// TwinCAT 3 PLC project CX5240
// ProgramVersion: 3.1.4026.13
// libraries:
//   CmpBitmapPool, * (System)
//   Tc2_Standard, * (Beckhoff Automation GmbH)
//   Tc2_System, * (Beckhoff Automation GmbH)
//   Tc3_Module, * (Beckhoff Automation GmbH)
//   VisuDialogs, * (System)
//   VisuSymbols,3.5.10.0,System
// project tree:
//   Enums/ E_Status.TcDUT (not stored)
//   Function Blocks/ FB_AnalogInputScaling.TcPOU (not stored), FB_DisplacementControl.TcPOU (not stored), FB_Encoder.TcPOU (not stored), FB_Integrator.TcPOU, FB_Joystick.TcPOU (not stored), FB_JoystickInputScaling.TcPOU (not stored), FB_DisplacementValveOutput.TcPOU (not stored), FB_StartPos.TcPOU, FB_YokeInputScaling.TcPOU (not stored), FB_ValveOutput.TcPOU
//   / GlobalTextList.TcGTLO (not stored), PlcTask.TcTTO (not stored)
//   GVLs/ G_IO.TcGVL (not stored), G_Parameters.TcGVL (not stored), G_Sensors.TcGVL (not stored), HMI.TcGVL
//   POUs/ MAIN.TcPOU, P_Inputs.TcPOU (not stored), P_MotionControl.TcPOU (not stored), P_Outputs.TcPOU
//   Struct/ ST_AnalogInputScaling.TcDUT (not stored), ST_JoystickInputScaling.TcDUT, ST_YokeInputScaling.TcDUT (not stored), ST_Parameters.TcDUT, ST_ValveDeadBand.TcDUT (not stored), ST_ValveOutput.TcDUT (not stored)
// real-time tasks:
//   TASK PlcTask: cycle T#1ms, priority 20, ADS port 350
//   TASK VISU_TASK: cycle T#200000us, priority 30, ADS port 351
// I/O:
//   DEVICE Device 1 (EtherCAT), AmsNetId 128.39.200.126.2.1
//     Term 1 (EK1200) [EK1200-5000 EtherCAT Power supply (2A E-Bus)]
//       Term 2 (EL1859) [EL1859 8Ch. Dig. Input 24V, 3ms, 8Ch. Dig. Output 24V, 0.5A]
//       Term 3 (EL3174) [EL3174 4Ch. Ana. Input +/-10V Diff., +/-20mA SingleEnded, 16 Bit]
//       Term 4 (EL4032) [EL4032 2Ch. Ana. Output +/-10V, 12bit]
//       Term 7 (EL3204) [EL3204 4Ch. Ana. Input PT100 (RTD)]
//       Term 8 (EK1110) [EK1110 EtherCAT extension]
//     Term 14 (EK1818) [EK1818 EtherCAT IO-Coupler  (1A E-Bus, 8 Ch. Dig. In, 3ms, 4 Ch. Dig. Out 24V, 0,5A)] (disabled)
//       Term 10 (EL1008) [EL1008 8Ch. Dig. Input 24V, 3ms]
//       Term 11 (EL3174) [EL3174 4Ch. Ana. Input +/-10V Diff., +/-20mA SingleEnded, 16 Bit]
//       Term 12 (EL3068) [EL3068 8Ch. Ana. Input 0-10V]
//       Term 5 (EL4032) [EL4032 2Ch. Ana. Output +/-10V, 12bit]
//       Term 6 (EL4122) [EL4122 2Ch. Ana. Output  4-20mA, 16bit]
//       Term 17 (EL9011) [EL9011 End Terminal]
//     Box 13 (Fraba EtherCAT) [Absolute Rotary Encoder IXARC V01.05] (disabled)
// variable links:
//   CX5240/CX5240 Instance <-> Device 1 (EtherCAT)/Term 1 (EK1200)/Term 2 (EL1859)
//     PlcTask Inputs/G_IO.bTestNew <-> Channel 1/Input
//   CX5240/CX5240 Instance <-> Device 1 (EtherCAT)/Term 14 (EK1818)
//     PlcTask Inputs/G_IO.bEmgOk <-> Channel 1/Input
//     PlcTask Outputs/G_IO.bEnablePCDV <-> Channel 10/Output
//     PlcTask Outputs/G_IO.bOpenBrakes <-> Channel 9/Output
//     PlcTask Outputs/G_IO.bWinchValveEnable <-> Channel 11/Output
//   CX5240/CX5240 Instance <-> Device 1 (EtherCAT)/Term 14 (EK1818)/Term 10 (EL1008)
//     PlcTask Inputs/G_IO.bAutoSwtich <-> Channel 3/Input
//     PlcTask Inputs/G_IO.bDisplacementEnable <-> Channel 7/Input
//     PlcTask Inputs/G_IO.bManualSwtich <-> Channel 1/Input
//     PlcTask Inputs/G_IO.bOffSwtich <-> Channel 2/Input
//     PlcTask Inputs/G_IO.bStartButton <-> Channel 4/Input
//     PlcTask Inputs/G_IO.bStopButton <-> Channel 5/Input
//     PlcTask Inputs/G_IO.bWinchEnable <-> Channel 6/Input
//   CX5240/CX5240 Instance <-> Device 1 (EtherCAT)/Term 14 (EK1818)/Term 11 (EL3174)
//     PlcTask Inputs/G_IO.fPDCVMonitor <-> AI Standard Channel 1/Value
//     PlcTask Inputs/G_IO.fPressureWinchB <-> AI Standard Channel 3/Value
//     PlcTask Inputs/G_IO.fYoke <-> AI Standard Channel 4/Value
//     PlcTask Inputs/G_IO.nMoogMonitor <-> AI Standard Channel 2/Value
//   CX5240/CX5240 Instance <-> Device 1 (EtherCAT)/Term 14 (EK1818)/Term 12 (EL3068)
//     PlcTask Inputs/G_IO.fJoyXraw <-> AI Standard Channel 6/Value
//     PlcTask Inputs/G_IO.fJoyYraw <-> AI Standard Channel 7/Value
//     PlcTask Inputs/G_IO.fJoyZraw <-> AI Standard Channel 8/Value
//     PlcTask Inputs/G_IO.fPressureReturn <-> AI Standard Channel 3/Value
//     PlcTask Inputs/G_IO.fPressureSupply <-> AI Standard Channel 2/Value
//     PlcTask Inputs/G_IO.fPressureWinchA <-> AI Standard Channel 1/Value
//   CX5240/CX5240 Instance <-> Device 1 (EtherCAT)/Term 14 (EK1818)/Term 5 (EL4032)
//     PlcTask Outputs/G_IO.fWinchPDCVOut <-> AO Outputs Channel 1/Analog output
//   CX5240/CX5240 Instance <-> Device 1 (EtherCAT)/Term 14 (EK1818)/Term 6 (EL4122)
//     PlcTask Outputs/G_IO.fWinchValveOut <-> Channel 1/Output

// ---- Struct/ST_JoystickInputScaling.TcDUT
TYPE ST_JoystickInputScaling :
STRUCT
	fMaxInputValue			: LREAL;	// tunable max input value
	fMinInputValue 			: LREAL;	// tunable min input value
	fNeutralInputValue  	: LREAL;	// tunable neutral input value
	fNeutralDeadband		: LREAL;	// tunable dead_band value
	fMaxOutputValue  		: LREAL;	// normalized max output value
	fMinOutputValue  		: LREAL;	// normalized min output value
	fNeutralOutputValue  	: LREAL;	// normalized neutral output value
END_STRUCT
END_TYPE

// ---- Struct/ST_Parameters.TcDUT
 TYPE ST_Parameters :
STRUCT
	fCyclicTime 					: LREAL := 0.001; // [s]
	fMaxWinchVelocityLimit 			: LREAL := 0.025; // [m/s]
	bWinchDeadBandCompOn 			: BOOL := FALSE;
	bDisplacementDeadBandCompOn 	: BOOL := FALSE;
	stWinchValveDeadBand 			: ST_ValveDeadBand := (fPosMax := 32767.0, fPosMin := 16383.0, fNegMin := 16383.0, fNegMax := 0);
	stDisplacementValveDeadBand 	: ST_ValveDeadBand := (fPosMax := 32767.0, fPosMin := 16383.0, fNegMin := 16383.0, fNegMax := 0);
	stPressureSensorScaling400bar 	: ST_AnalogInputScaling := (fMaxInputValue := 32767.0, fMinInputValue := 0.0, fMaxOutputValue := 400.0, fMinOutputValue := 0.0);
	stPressureSensorScaling40bar 	: ST_AnalogInputScaling := (fMaxInputValue := 32767.0, fMinInputValue := 0.0, fMaxOutputValue := 40.0, fMinOutputValue := 0.0);
	stJoystickInputScalingX 		: ST_JoystickInputScaling := (fMaxInputValue := 14790.0, fMinInputValue := 1797.0, fNeutralInputValue := 8400, fNeutralDeadband := 50.0, fMaxOutputValue := 1.0, fMinOutputValue := -1.0, fNeutralOutputValue := 0.0);
	stJoystickInputScalingY 		: ST_JoystickInputScaling := (fMaxInputValue := 14770.0, fMinInputValue := 1829.0, fNeutralInputValue := 8340, fNeutralDeadband := 50.0, fMaxOutputValue := 1.0, fMinOutputValue := -1.0, fNeutralOutputValue := 0.0);
	stJoystickInputScalingZ 		: ST_JoystickInputScaling := (fMaxInputValue := 14830.0, fMinInputValue := 1804.0, fNeutralInputValue := 8380, fNeutralDeadband := 50.0, fMaxOutputValue := 1.0, fMinOutputValue := -1.0, fNeutralOutputValue := 0.0);
	fWinchEncoderOffset 			: LREAL := -5886686.1725795381; // Encoder value at zero (Cylinder out / second layaer)
	stYokeInputScaling 				: ST_YokeInputScaling := (fMaxInputValue := 25000.0, fMinInputValue := 6150.0, fNeutralInputValue := 15470, fNeutralDeadband := 0.0, fMaxOutputValue := 1.0, fMinOutputValue := -1.0, fNeutralOutputValue := 0.0);
	fWinchDrumRadius 				: LREAL := 0.075;
	fWinchEndStopPos 				: LREAL := 2.16;
	fWinchEndStopNeg 				: LREAL := 1.0;
	fPayloadMass 					: LREAL := 78.0; 
END_STRUCT
END_TYPE

// ---- GVLs/HMI.TcGVL
{attribute 'qualified_only'}
VAR_GLOBAL
	bEndStopOverride : BOOL; 
END_VAR

// ---- Function Blocks/FB_Integrator.TcPOU
FUNCTION_BLOCK FB_Integrator
VAR_INPUT
	ssMethodType: SINT;
	bEnable: BOOL;
	VelRef_ms: LREAL;
	PosInit_m: LREAL;
END_VAR
VAR_OUTPUT
	PosRef_m: LREAL;
END_VAR
VAR
	c_DiscreteTimeIntegrator_IC: USINT;
	c_DiscreteTimeIntegrator_DS: LREAL;
END_VAR



CASE ssMethodType OF
    0: 
        (* SystemInitialize for Atomic SubSystem: '<Root>/FB_Integrator' *)
        (* InitializeConditions for DiscreteIntegrator: '<S1>/Discrete-Time Integrator' *)
        c_DiscreteTimeIntegrator_IC := 1;
        (* End of SystemInitialize for SubSystem: '<Root>/FB_Integrator' *)
    1: 
        (* Outputs for Atomic SubSystem: '<Root>/FB_Integrator' *)
        (* DiscreteIntegrator: '<S1>/Discrete-Time Integrator' *)

        IF c_DiscreteTimeIntegrator_IC <> 0 THEN 
            c_DiscreteTimeIntegrator_DS := PosInit_m;
        END_IF;

        (* Switch: '<S1>/Switch' *)

        IF bEnable THEN 
            (* Outport: '<Root>/PosRef_m' incorporates:
             *  DiscreteIntegrator: '<S1>/Discrete-Time Integrator' *)
            PosRef_m := c_DiscreteTimeIntegrator_DS;
        ELSE 
            (* Outport: '<Root>/PosRef_m' *)
            PosRef_m := PosInit_m;
        END_IF;

        (* End of Switch: '<S1>/Switch' *)
        

        (* Update for DiscreteIntegrator: '<S1>/Discrete-Time Integrator' *)
        c_DiscreteTimeIntegrator_IC := 0;
        c_DiscreteTimeIntegrator_DS := (0.01 * VelRef_ms) + c_DiscreteTimeIntegrator_DS;
        (* End of Outputs for SubSystem: '<Root>/FB_Integrator' *)
END_CASE;

END_FUNCTION_BLOCK

// ---- Function Blocks/FB_StartPos.TcPOU
FUNCTION_BLOCK FB_StartPos
VAR_INPUT
	bEnable 		: BOOL;
	fCurrentPos 	: LREAL;
END_VAR
VAR_OUTPUT
	fStartPos 		: LREAL;
END_VAR
VAR
END_VAR

IF bEnable THEN
	fStartPos := fStartPos;
	
ELSE 
	fStartPos := fCurrentPos;
END_IF

END_FUNCTION_BLOCK

// ---- Function Blocks/FB_ValveOutput.TcPOU
FUNCTION_BLOCK FB_ValveOutput
VAR_INPUT
	bEnable 			: BOOL;
	bDeadBandCompOn 	: BOOL;
	stValveDeadBand 	: ST_ValveDeadBand;
	fNormalizedInput 	: LREAL;
END_VAR
VAR_OUTPUT
	bEnableValveOutput : BOOL;
	nOutput : INT; 
END_VAR
VAR
	nOffset 	: INT := 16383;
	nMaxValue	: INT := 20000;
	nMinValue 	: INT :=  12766;
	nTempOutput : INT := 16383;
END_VAR

IF	bDeadBandCompOn THEN
	IF fNormalizedInput > 0.0 THEN
		nTempOutput := LREAL_TO_INT(ABS(fNormalizedInput*(stValveDeadBand.fPosMax - stValveDeadBand.fPosMin) + stValveDeadBand.fPosMin));
	ELSIF fNormalizedInput < 0.0 THEN
		nTempOutput := LREAL_TO_INT(ABS(fNormalizedInput*(stValveDeadBand.fNegMax - stValveDeadBand.fNegMin) - stValveDeadBand.fNegMin));
	ELSE
		nTempOutput := nOffset;
	END_IF
ELSE
	IF fNormalizedInput > 0.0  THEN
		nTempOutput := LREAL_TO_INT(ABS(fNormalizedInput*(32767.0 - 16383.0) + 16383.0));
	ELSIF fNormalizedInput < 0.0  THEN
		nTempOutput := LREAL_TO_INT(ABS(fNormalizedInput*(0 - 16383.0) - 16383.0));
	ELSE
		nTempOutput := nOffset;
	END_IF	
END_IF		



IF bEnable THEN
	nOutput := LIMIT(nMinValue, nTempOutput, nMaxValue);
	bEnableValveOutput := TRUE; 
ELSE 	
	nOutput := nOffset;
	bEnableValveOutput := FALSE;	
END_IF

END_FUNCTION_BLOCK

// ---- POUs/MAIN.TcPOU
PROGRAM MAIN
VAR
	bStatusOk : BOOL;
	bFault : BOOL := FALSE;
	eStatus : E_Status := E_Status.Checking;
	bRunning : BOOL := TRUE;
END_VAR

P_Inputs();
P_Outputs();
P_MotionControl();
	
// State Machine for selecting mode
IF G_IO.bEmgOk AND NOT(G_IO.bStopButton) AND NOT(G_IO.bOffSwtich) AND NOT(bFault) THEN
	bStatusOk := TRUE;
ELSE 
	bStatusOk := FALSE;
END_IF

CASE eStatus OF 
	E_Status.Checking:
		IF bFault THEN
			eStatus := E_Status.Fault;
		END_IF
		
		IF bStatusOk THEN	
			eStatus := E_Status.Ready;
		END_IF
		
		IF NOT(bStatusOk) THEN	
			eStatus := E_Status.Off;
		END_IF
		
	E_Status.Off:	
		IF bStatusOk THEN	
			eStatus := E_Status.Checking;
		END_IF
		
		IF bFault THEN
			eStatus := E_Status.Fault;
		END_IF

	E_Status.Fault:
		IF NOT(bFault) THEN
			eStatus := E_Status.Checking;
		END_IF
	
	E_Status.Ready:
		IF G_IO.bStartButton AND bStatusOk AND NOT(bFault) THEN
			eStatus := E_Status.Starting;
		END_IF	
		
		IF  NOT(bStatusOk) OR bFault THEN
			eStatus := E_Status.Checking;
		END_IF	

	E_Status.Starting:
		IF bRunning THEN
			eStatus := E_Status.Running;
		END_IF 
		
		IF bFault OR NOT(bStatusOk)  THEN
			eStatus := E_Status.Checking;
		END_IF
			
	E_Status.Running:
		IF G_IO.bStopButton THEN
			eStatus := E_Status.Stopping;
		END_IF
		
		IF NOT(bRunning) OR NOT(bStatusOk) OR bFault THEN
			eStatus := E_Status.Checking;
		END_IF
	
	E_Status.Stopping:	
		IF NOT(bRunning) THEN
			eStatus := E_Status.Checking;
		END_IF
	
		IF NOT(bStatusOk) OR bFault THEN
		eStatus := E_Status.Checking;
		END_IF	
	
ELSE 	
	eStatus := E_Status.Checking;
END_CASE

END_PROGRAM

// ---- POUs/P_Outputs.TcPOU
PROGRAM P_Outputs
VAR
	fbWinchValveOutput 				: FB_ValveOutput;
	fbDisplacementValveOutput 		: FB_DisplacementValveOutput;
	eStatus 						: E_Status; 
	bEnableWinch 					: BOOL;
	bEnableDisplacement 			: BOOL;
	fDisplacementControlSignal  	: LREAL;
	fDisplacementNormalizedInput 	: LREAL := 1.0;
	bEndStopNegActive 				: BOOL;
	bEndStopPosActive 				: BOOL;
	fWinchValveNormalizedInput  	: LREAL;
	fWinchValveInput 				: LREAL;
	bEnableMotion 					: BOOL;	
	bEnableValveOutputWinch 		: BOOL; 
	bEnableValveOutputDisp	 		: BOOL; 
END_VAR

IF MAIN.eStatus = E_Status.Running THEN
	G_IO.bEnablePCDV := TRUE;
	G_IO.bWinchValveEnable := TRUE;
ELSE
	G_IO.bEnablePCDV := FALSE;	
	G_IO.bWinchValveEnable := FALSE;
END_IF

bEnableMotion := G_IO.bWinchEnable;

///////////////////// Winch //////////////////////////////
IF (MAIN.eStatus = E_Status.Running) AND bEnableMotion THEN 
	G_IO.bOpenBrakes := TRUE;
	bEnableWinch := TRUE;
ELSE
	G_IO.bOpenBrakes := FALSE;
	bEnableWinch := FALSE;
END_IF

///////////////////// Displacement //////////////////////////////
IF (MAIN.eStatus = E_Status.Running) AND G_IO.bDisplacementEnable THEN 
	bEnableDisplacement := TRUE;
ELSE
	bEnableDisplacement := FALSE;
END_IF

fWinchValveInput := G_Sensors.fJoystickNormalizedY;

IF P_MotionControl.fWinchPos < G_Parameters.stParam.fWinchEndStopNeg  AND NOT(HMI.bEndStopOverride) THEN
	bEndStopPosActive := FALSE;
	bEndStopNegActive := TRUE;
	fWinchValveNormalizedInput := LIMIT(-1.0, fWinchValveInput, 0.0);
ELSIF P_MotionControl.fWinchPos > G_Parameters.stParam.fWinchEndStopPos AND NOT(HMI.bEndStopOverride) THEN
	bEndStopPosActive := TRUE;
	bEndStopNegActive := FALSE;
	fWinchValveNormalizedInput := LIMIT(0, fWinchValveInput, 1.0);
ELSE
	bEndStopPosActive := FALSE;
	bEndStopNegActive := FALSE;
	fWinchValveNormalizedInput := fWinchValveInput;
END_IF

fbWinchValveOutput(
	bEnable := bEnableWinch,
	bDeadBandCompOn := G_Parameters.stParam.bWinchDeadBandCompOn,
	stValveDeadBand := G_Parameters.stParam.stWinchValveDeadBand,
	fNormalizedInput := fWinchValveNormalizedInput,
	bEnableValveOutput => bEnableValveOutputWinch,
	nOutput => G_IO.fWinchValveOut
);

IF NOT(bEnableDisplacement) THEN
	fDisplacementControlSignal := fDisplacementNormalizedInput; 
ELSE	
	fDisplacementControlSignal := G_Sensors.fJoystickNormalizedZ;
END_IF

fbDisplacementValveOutput(
	bEnable := (MAIN.eStatus = E_Status.Running),
	bDeadBandCompOn := G_Parameters.stParam.bDisplacementDeadBandCompOn,
	stValveDeadBand := G_Parameters.stParam.stDisplacementValveDeadBand,
	fNormalizedInput := fDisplacementControlSignal,
	bEnableValveOutput => bEnableValveOutputDisp,
	nOutput => G_IO.fWinchPDCVOut
);

END_PROGRAM
